// TIA Portal project "1200 Modbus TCP" (V20)

(* hardware
DEVICE "S7-1200 station_1"  S7-1200 Station
   slot 0: "Rack_0"  S7-1200 Rack  Rack  V1.0
   slot 1: "PLC_1"  CPU 1215C DC/DC/DC  6ES7 215-1AG40-0XB0  V4.6
   slot 3: "CB 1241 (RS485)"  CB 1241 (RS485)  6ES7 241-1CH30-1XB0  V1.0
*)

// ===== PLC "PLC_1"  CPU 1215C DC/DC/DC =====

VAR_GLOBAL   // PLC tag table "Default tag table"
   "桌面丝杆_Pulse" AT %Q0.0 : Bool;
   "桌面丝杆_Direction" AT %Q0.2 : Bool;
   "桌面丝杆_LowHwLimitSwitch" AT %I0.0 : Bool;
   "桌面丝杆_HighHwLimitSwitch" AT %I0.2 : Bool;
   "桌面丝杆_Homing switch" AT %I0.1 : Bool;
   "Tag_1" AT %I0.3 : Bool;
   "Tag_2" AT %Q0.1 : Bool;
   "Tag_3" AT %Q0.3 : Bool;
   "Tag_4" AT %Q0.4 : Bool;
   "Tag_5" AT %Q0.5 : Bool;
   "Tag_6" AT %Q0.6 : Bool;
   "Tag_7" AT %Q0.7 : Bool;
   "Tag_8" AT %Q1.0 : Bool;
   "Tag_9" AT %Q1.1 : Bool;
   "Tag_10" AT %Q1.2 : Bool;
   "Tag_11" AT %Q1.3 : Bool;
   "Tag_12" AT %Q1.4 : Bool;
   "Tag_13" AT %Q1.5 : Bool;
   "Tag_14" AT %Q1.6 : Bool;
   "Tag_15" AT %Q1.7 : Bool;
   "Tag_16" AT %Q2.0 : Bool;
   "Tag_17" AT %Q2.1 : Bool;
   "Tag_18" AT %Q2.2 : Bool;
   "Tag_19" AT %Q2.3 : Bool;
   "Tag_20" AT %Q2.4 : Bool;
   "Tag_21" AT %Q2.5 : Bool;
   "Tag_22" AT %Q2.6 : Bool;
   "Tag_23" AT %Q2.7 : Bool;
   "hmi1" AT %QB0 : Byte;
END_VAR

DATA_BLOCK "Block_1_DB"   // DB2
{ S7_Optimized_Access := 'FALSE' }
VERSION : 0.1
// stored: InstanceOfName Block_1
"Block_1"
BEGIN
END_DATA_BLOCK

DATA_BLOCK "Db Global"   // DB3
{ S7_Optimized_Access := 'TRUE' }
VERSION : 0.1
   VAR
      connection : TCON_IP_v4;
   END_VAR
BEGIN
   connection.InterfaceId := 64;
   connection.ID := 1;
   connection.LocalPort := 502;
END_DATA_BLOCK

FUNCTION_BLOCK "Block_1"   // FB2, SCL
{ S7_Optimized_Access := 'FALSE' }
VERSION : 0.1
   VAR
      value1 : Word;
      value2 : Word;
      value3 : Word;
      value4 : Word;
      value5 : Word;
      value6 : Word;
      value7 : Word;
      value8 : Word;
      value9 : Word;
      value10 : Word;
      value11 : Word;
      value12 : Word;
      value13 : Word;
      value14 : Word;
      value15 : Word;
      value16 : Word;
      value17 : Word;
      value18 : Word;
      value19 : Word;
      value20 : Word;
      value21 : Word;
      value22 : Word;
      value23 : Word;
      value24 : Word;
      value25 : Word;
      value26 : Word;
      value27 : Word;
      value28 : Word;
      value29 : Word;
      value30 : Word;
   END_VAR
BEGIN
END_FUNCTION_BLOCK

ORGANIZATION_BLOCK "Main"   // OB1, LAD, ProgramCycle
TITLE = "Main Program Sweep (Cycle)"
{ S7_Optimized_Access := 'TRUE' }
VERSION : 0.1
   VAR_INPUT
      Initial_Call : Bool;   // Initial call of this OB
      Remanence : Bool;   // =True, if remanent data are available
   END_VAR
BEGIN

REGION Network 1
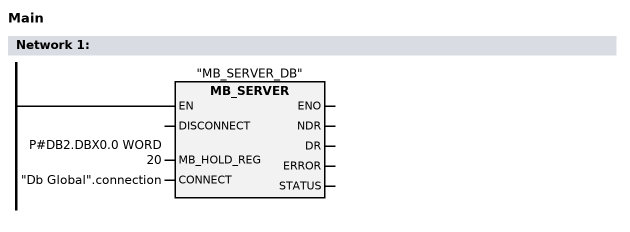
   "MB_SERVER_DB"(MB_HOLD_REG := P#DB2.DBX0.0 WORD 20, CONNECT := "Db Global".connection);   // MB_SERVER
END_REGION
END_ORGANIZATION_BLOCK